# EPICS substitutions: Lakeshore340Sup/Lakeshore340_channel.substitutions
file Lakeshore340_channel.template {

  pattern {PORT, P, CHAN, SENS_NUM}
  {"\$(PORT)", "\$(P)", "A", "0"}
  {"\$(PORT)", "\$(P)", "B", "1"}
  {"\$(PORT)", "\$(P)", "C", "2"}
  {"\$(PORT)", "\$(P)", "D", "3"}
}
